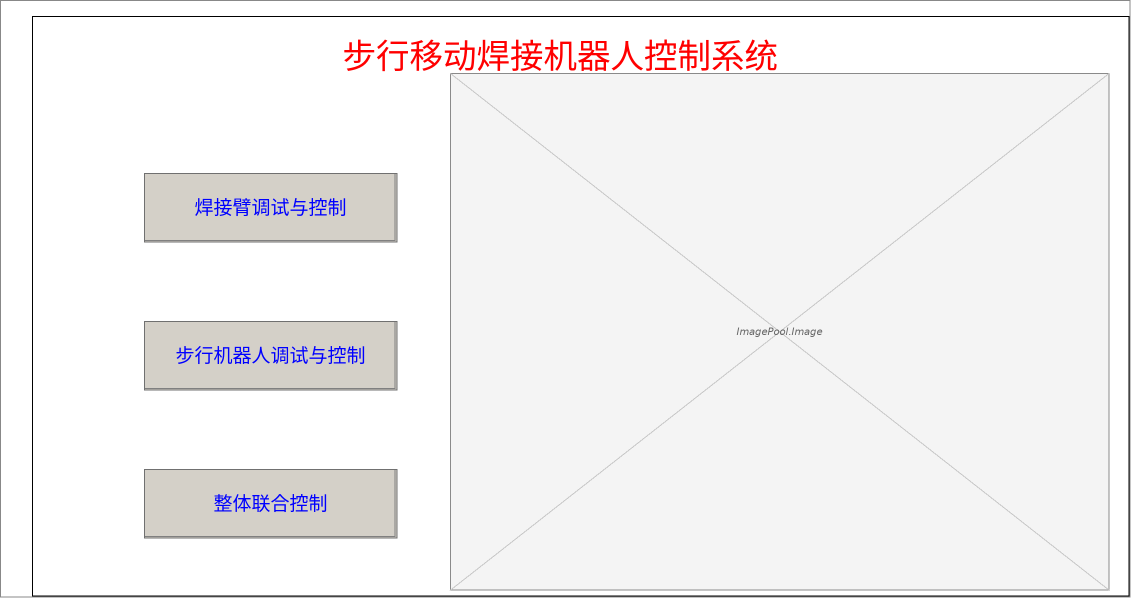
VISUALIZATION Visu_Welcome  // 1131x598
    Rectangle (32,16 1097x580)
    Image (716,328 150x30)
    Label (269,35 583x42), "步行移动焊接机器人控制系统"
    Button (144,469 253x69), "整体联合控制"
        OnMouseClick: change screen: Visu_Walking_Welding_Robot_Control
    Button (144,321 253x69), "步行机器人调试与控制"
        OnMouseClick: change screen: Visu_Walking_Robot_Power
    Button (144,173 253x69), "焊接臂调试与控制"
        OnMouseClick: change screen: Visu_Welding_Arm_Power
    Image (450,73 659x517), image: ImagePool.Image
END_VISUALIZATION

(* stored: Version 1.1.0.1, ProductVersion 3.1.4020.12
   Visu Visu_Welcome: Id {d13f4a69-5f56-48ce-899e-695870ed65dd} *)
